FUNCTION_BLOCK PAMBeltscale EXTENDS PAProcessModule
VAR_INPUT
END_VAR
VAR_OUTPUT
END_VAR
VAR
	_PAPointMatIn1 : PAPoint(THIS^);
	_PAPointMatOut1 : PAPoint(THIS^);
END_VAR

METHOD FB_init : BOOL
VAR_INPUT
	bInitRetains : BOOL; // if TRUE, the retain variables are initialized (warm start / cold start)
	bInCopyCode : BOOL;  // if TRUE, the instance afterwards gets moved into the copy code (online change)
	parent : IACComponent;
END_VAR
AddPoint(_PAPointMatIn1);
AddPoint(_PAPointMatOut1);
END_METHOD

PROPERTY PUBLIC PAPointMatIn1 : IACPoint
GET
PAPointMatIn1 := _PAPointMatIn1;
END_GET
END_PROPERTY

PROPERTY PUBLIC PAPointMatOut1 : IACPoint
GET
PAPointMatOut1 := _PAPointMatOut1;
END_GET
END_PROPERTY

END_FUNCTION_BLOCK

(* stored: Version 1.1.0.1, ProductVersion 3.1.4020.12
   POU PAMBeltscale: Id {f6ee7a6b-bcfc-4fd3-9cc2-51ca2a032c8c}, SpecialFunc None
   Method FB_init: Id {731da9fd-4add-4430-9f30-fe5c757b9fa8}
   Property PAPointMatIn1: Id {52b595c5-a241-400a-9fb2-8e74d25ee83f}
   Get Get: Id {b4a6e885-7b31-4280-8971-7dfc5fc3ab4d}
   Property PAPointMatOut1: Id {6f87d9e5-be8e-4a12-a0c8-bf0776b1a812}
   Get Get: Id {20c9679a-27c6-459f-90bf-f357c7f54465} *)
